TYPE HLSInputData_1 :
STRUCT
	//In
	iIn : INT;
	
	//Out
	iOut : INT;
END_STRUCT
END_TYPE

(* stored: Version 1.1.0.1, ProductVersion 3.1.4024.12
   DUT HLSInputData_1: Id {e30c512b-1a91-4ccd-a1f3-93fa3eeb07a2} *)
